// TIA Portal V17 export
// export: Created 2023-09-10T16:27:50.0847162Z, ExportSetting WithDefaults, DisplayName Totally Integrated Automation Portal, DisplayVersion V17, DisplayName TIA Portal Openness, DisplayVersion V17, DisplayName TIA Portal Version Control Interface, DisplayVersion V17, DisplayName STEP 7 Professional, DisplayVersion V17, DisplayName STEP 7 Safety, DisplayVersion V17, DisplayName WinCC Advanced, DisplayVersion V17
FUNCTION "modbusEncoder" : Void   // FC1, LAD
{ S7_Optimized_Access := 'TRUE' }
VERSION : 0.1
// stored: AutoNumber true, IsIECCheckEnabled false, SetENOAutomatically false, UDAEnableTagReadback false
   VAR_INPUT
      encoderModbusAdress : UInt;
      modbusMode : USInt;   // modbus mode; 0- read holding register(03);1-Writing a holding register; see help MB_Master
      dataAddress : UDInt;   // starting adress (40001)
      dataLength : UDInt;
      encoderValue : Int;
      maxEncoderValue : Int;
      firstScanBit : Bool;
   END_VAR
   VAR_OUTPUT
      mbStatusWord : Word;
   END_VAR
   VAR_IN_OUT
      lastEncoderValue : Int;
      machinePosition : DInt;
      turn : DInt;
      mbBusyBit : Bool;
      mbDoneBit : Bool;
      mbErrorBit : Bool;
      mbReq : Bool;
      mbAgain : Bool;
      "timer" : IEC_TIMER;
   END_VAR
   VAR_TEMP
      rotationDistance : DInt;
   END_VAR
BEGIN

REGION Network 1: Modbus data block
   // Pobranie danych po modbusie do bloku danych
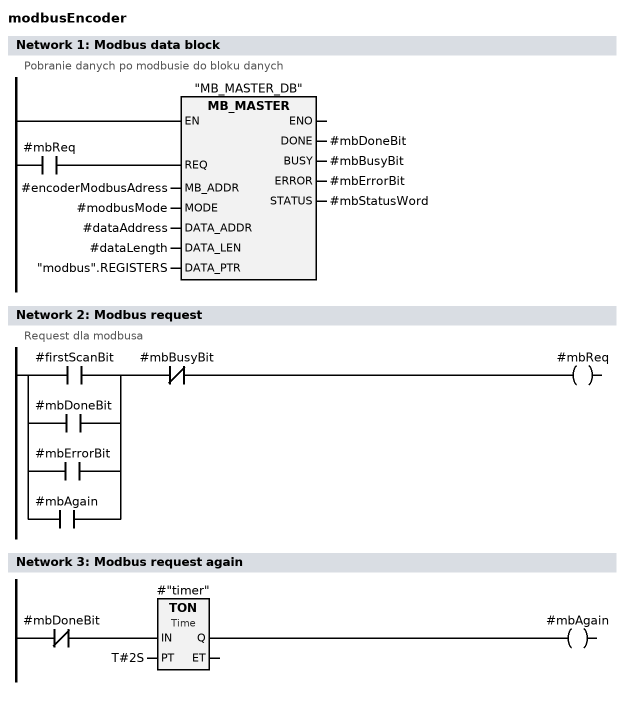
   RUNG wire#powerrail
      "MB_MASTER_DB".MB_MASTER(REQ := wire#w1, MB_ADDR := #encoderModbusAdress, MODE := #modbusMode, DATA_ADDR := #dataAddress, DATA_LEN := #dataLength, DATA_PTR := "modbus".REGISTERS, DONE => #mbDoneBit, BUSY => #mbBusyBit, ERROR => #mbErrorBit, STATUS => #mbStatusWord)
   END_RUNG
   RUNG wire#powerrail
      Contact( #mbReq )
   END_RUNG wire#w1
   // the same network as SCL:
   "MB_MASTER_DB"(REQ := #mbReq,   // MB_MASTER
                  MB_ADDR := #encoderModbusAdress,
                  MODE := #modbusMode,
                  DATA_ADDR := #dataAddress,
                  DATA_LEN := #dataLength,
                  DATA_PTR := "modbus".REGISTERS,
                  DONE => #mbDoneBit,
                  BUSY => #mbBusyBit,
                  ERROR => #mbErrorBit,
                  STATUS => #mbStatusWord);
END_REGION

REGION Network 2: Modbus request
   // Request dla modbusa
   RUNG wire#powerrail
      Contact( #firstScanBit )
      wire#w1
      I_Contact( #mbBusyBit )
      Coil( #mbReq )
   END_RUNG
   RUNG wire#powerrail
      Contact( #mbDoneBit )
   END_RUNG wire#w1
   RUNG wire#powerrail
      Contact( #mbErrorBit )
   END_RUNG wire#w1
   RUNG wire#powerrail
      Contact( #mbAgain )
   END_RUNG wire#w1
   // the same network as SCL:
   #mbReq := (#firstScanBit OR #mbDoneBit OR #mbErrorBit OR #mbAgain) AND NOT #mbBusyBit;
END_REGION

REGION Network 3: Modbus request again
   RUNG wire#powerrail
      I_Contact( #mbDoneBit )
      { S7_Templates := "time_type := Time" } #"timer".TON(pt := T#2S, et =>)
      Coil( #mbAgain )
   END_RUNG
   // the same network as SCL:
   #"timer".TON(IN := NOT #mbDoneBit, PT := T#2S);
   #mbAgain := #"timer".Q;
END_REGION

REGION Network 4 (SCL)
   #encoderValue := "modbus".REGISTERS[0];
   IF (#encoderValue <> #lastEncoderValue) THEN
       #rotationDistance := #encoderValue - #lastEncoderValue;
       IF (#rotationDistance > (#maxEncoderValue / 2)) THEN
           #turn := #turn - 1;
       ELSIF (#rotationDistance < ((-1) * #maxEncoderValue / 2)) THEN
           #turn := #turn + 1;
       END_IF;

       #machinePosition := #turn * #maxEncoderValue + #encoderValue;
       #lastEncoderValue := #encoderValue;

   END_IF;
END_REGION
END_FUNCTION
